INTERFACE I_IlluminationController_StatusOnly EXTENDS  __SYSTEM.IQueryInterface

{attribute 'monitoring' := 'call'}
PROPERTY Busy : BOOL
GET
END_GET
END_PROPERTY

{attribute 'monitoring' := 'call'}
PROPERTY Operational : BOOL
GET
END_GET
END_PROPERTY

{attribute 'monitoring' := 'call'}
PROPERTY PUBLIC State : E_StateTerminal
GET
END_GET
END_PROPERTY

END_INTERFACE

(* stored: Version 1.1.0.1, ProductVersion 3.1.4024.12
   Itf I_IlluminationController_StatusOnly: Id {6df00ed0-934e-4040-8eba-8c3512cabfb7}
   Property Busy: Id {f23de217-6599-414c-ba8d-f091e9759a5f}
   Get Get: Id {cf3a3cf9-6779-4390-a192-5c40268ef192}
   Property Operational: Id {5a09df8e-e8fc-4e4a-9a48-58a9d961aa5f}
   Get Get: Id {9ab958d2-ac5b-451e-8aad-91e3186d7dc5}
   Property State: Id {543a09c5-ab31-4332-b529-99608eba5752}
   Get Get: Id {d5405189-e9c5-4fcb-907b-785e9414ab9d} *)
